FUNCTION_BLOCK Voltage EXTENDS SM_Voltage
VAR_INPUT
END_VAR
VAR_OUTPUT
END_VAR
VAR
    _testVar : INT;
END_VAR

SUPER^();

END_FUNCTION_BLOCK

(* stored: Version 1.1.0.1, ProductVersion 3.1.4018.2
   POU Voltage: Id {def5fc12-e190-4589-a260-3267dfd7fe2e}, SpecialFunc None *)
